Staubli VAL3: start.pgx

program start()
begin
  cls()
  movej(JHome,tTool, mNomSpeed)
  waitEndMove()
  movej(JApproach1,tTool, mNomSpeed)
  waitEndMove()
  do
    // Leo caracter
    clearBuffer(sSioOrdenador)
    delay(5)
    nTest = sioGet(sSioOrdenador, l_nNumero)
    put("Test :")
    put(nTest)
    put(" L_nNumero :")
    put(l_nNumero)
    putln(" ")

    sioSet(sSioOrdenador, l_nNumero)


  until l_nNumero == 13
end
